{attribute addProperty BoxType "EM3702-0000-0016"}
{attribute addProperty Id "StatusAT %I*Status_3D195A321621ValueAT %I*INT16217"}
{attribute addProperty CRC "3613813698"}
{attribute addProperty SizeInBites "32"}
{attribute addProperty SizeInBytes "4"}
TYPE AI_Input_Channel_D7666BC2 :
STRUCT
	{attribute addProperty Name "Status"}
	Status AT %I* : Status_3D195A32;
	{attribute addProperty Name "Value"}
	Value AT %I* : INT;
END_STRUCT
END_TYPE

(* stored: Version 1.2.0.0, ProductVersion 3.1.4024.9
   DUT AI_Input_Channel_D7666BC2: Id {138348ac-197d-454c-9a22-fe03346cedb0} *)
